// TIA Portal V18 export
FUNCTION "Ratio Check Program sequences" : Void   // FC6, LAD
{ S7_Optimized_Access := 'TRUE' }
VERSION : 0.1
// stored: AutoNumber true, IsIECCheckEnabled false, SetENOAutomatically false, UDAEnableTagReadback false
   VAR_TEMP
      temp1 : Bool;
   END_VAR
   VAR_TEMP   // added for the SCL form of the ladder/FBD networks
      _w1 : Bool;
      _w2 : Bool;
      _w3 : Bool;
      _w4 : Bool;
   END_VAR
BEGIN

REGION Network 1
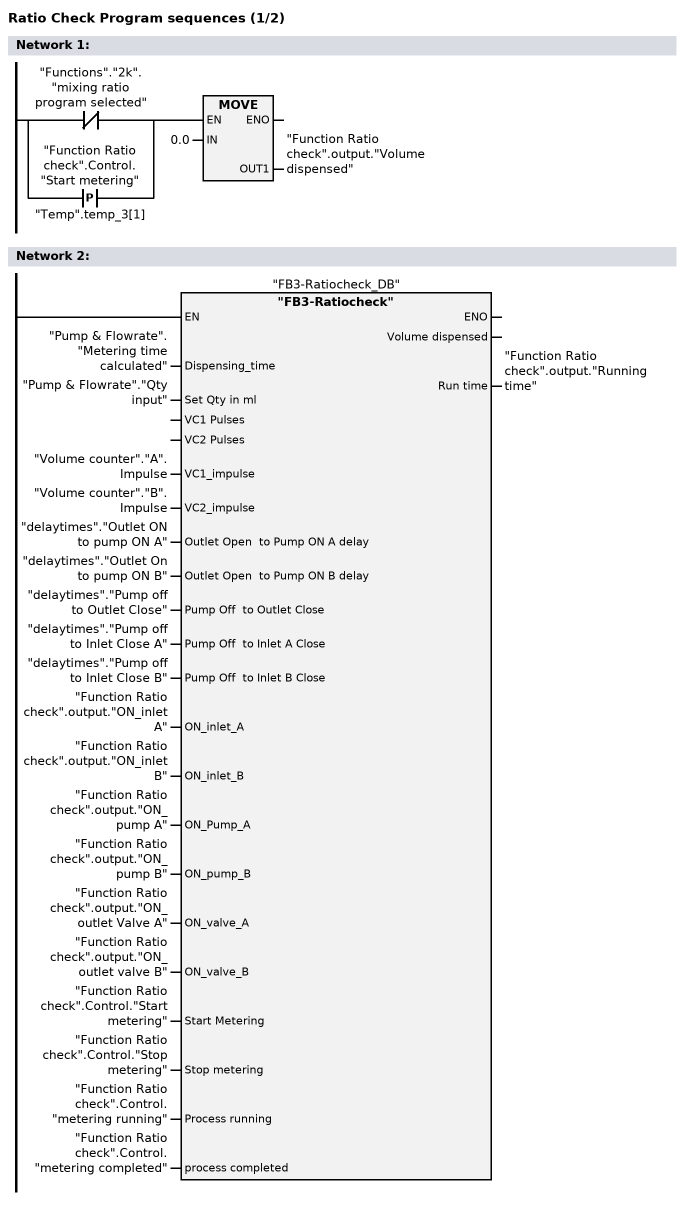
   RUNG wire#powerrail
      I_Contact( "Functions"."2k"."mixing ratio program selected" )
      wire#w1
      Move(in := 0.0, out1 => "Function Ratio check".output."Volume dispensed")
   END_RUNG
   RUNG wire#powerrail
      P_Contact(operand := "Function Ratio check".Control."Start metering", bit := "Temp".temp_3[1])
   END_RUNG wire#w1
   // the same network as SCL:
   #_w1 := "Function Ratio check".Control."Start metering" AND NOT "Temp".temp_3[1];   // rising edge of "Function Ratio check".Control."Start metering"
   "Temp".temp_3[1] := "Function Ratio check".Control."Start metering";
   IF NOT "Functions"."2k"."mixing ratio program selected" OR #_w1 THEN
       "Function Ratio check".output."Volume dispensed" := 0.0;
   END_IF;
END_REGION

REGION Network 2
   RUNG wire#powerrail
      "FB3-Ratiocheck_DB"(Dispensing_time := "Pump & Flowrate"."Metering time calculated", "Set Qty in ml" := "Pump & Flowrate"."Qty input", "VC1 Pulses" :=, "VC2 Pulses" :=, VC1_impulse := "Volume counter"."A".Impulse, VC2_impulse := "Volume counter"."B".Impulse, "Outlet Open  to Pump ON A delay" := "delaytimes"."Outlet ON to pump ON A", "Outlet Open  to Pump ON B delay" := "delaytimes"."Outlet On to pump ON B", "Pump Off  to Outlet Close" := "delaytimes"."Pump off to Outlet Close", "Pump Off  to Inlet A Close" := "delaytimes"."Pump off to Inlet Close A", "Pump Off  to Inlet B Close" := "delaytimes"."Pump off to Inlet Close B", ON_inlet_A := "Function Ratio check".output."ON_inlet A", ON_inlet_B := "Function Ratio check".output."ON_inlet B", ON_Pump_A := "Function Ratio check".output."ON_pump A", ON_pump_B := "Function Ratio check".output."ON_pump B", ON_valve_A := "Function Ratio check".output."ON_outlet Valve A", ON_valve_B := "Function Ratio check".output."ON_outlet valve B", "Start Metering" := "Function Ratio check".Control."Start metering", "Stop metering" := "Function Ratio check".Control."Stop metering", "Process running" := "Function Ratio check".Control."metering running", "process completed" := "Function Ratio check".Control."metering completed", "Volume dispensed" =>, "Run time" => "Function Ratio check".output."Running time")
   END_RUNG
   // the same network as SCL:
   "FB3-Ratiocheck_DB"(Dispensing_time := "Pump & Flowrate"."Metering time calculated",   // "FB3-Ratiocheck"
                       "Set Qty in ml" := "Pump & Flowrate"."Qty input",
                       VC1_impulse := "Volume counter"."A".Impulse,
                       VC2_impulse := "Volume counter"."B".Impulse,
                       "Outlet Open  to Pump ON A delay" := "delaytimes"."Outlet ON to pump ON A",
                       "Outlet Open  to Pump ON B delay" := "delaytimes"."Outlet On to pump ON B",
                       "Pump Off  to Outlet Close" := "delaytimes"."Pump off to Outlet Close",
                       "Pump Off  to Inlet A Close" := "delaytimes"."Pump off to Inlet Close A",
                       "Pump Off  to Inlet B Close" := "delaytimes"."Pump off to Inlet Close B",
                       ON_inlet_A := "Function Ratio check".output."ON_inlet A",
                       ON_inlet_B := "Function Ratio check".output."ON_inlet B",
                       ON_Pump_A := "Function Ratio check".output."ON_pump A",
                       ON_pump_B := "Function Ratio check".output."ON_pump B",
                       ON_valve_A := "Function Ratio check".output."ON_outlet Valve A",
                       ON_valve_B := "Function Ratio check".output."ON_outlet valve B",
                       "Start Metering" := "Function Ratio check".Control."Start metering",
                       "Stop metering" := "Function Ratio check".Control."Stop metering",
                       "Process running" := "Function Ratio check".Control."metering running",
                       "process completed" := "Function Ratio check".Control."metering completed",
                       "Run time" => "Function Ratio check".output."Running time");
END_REGION

REGION Network 3: Volume dispensed
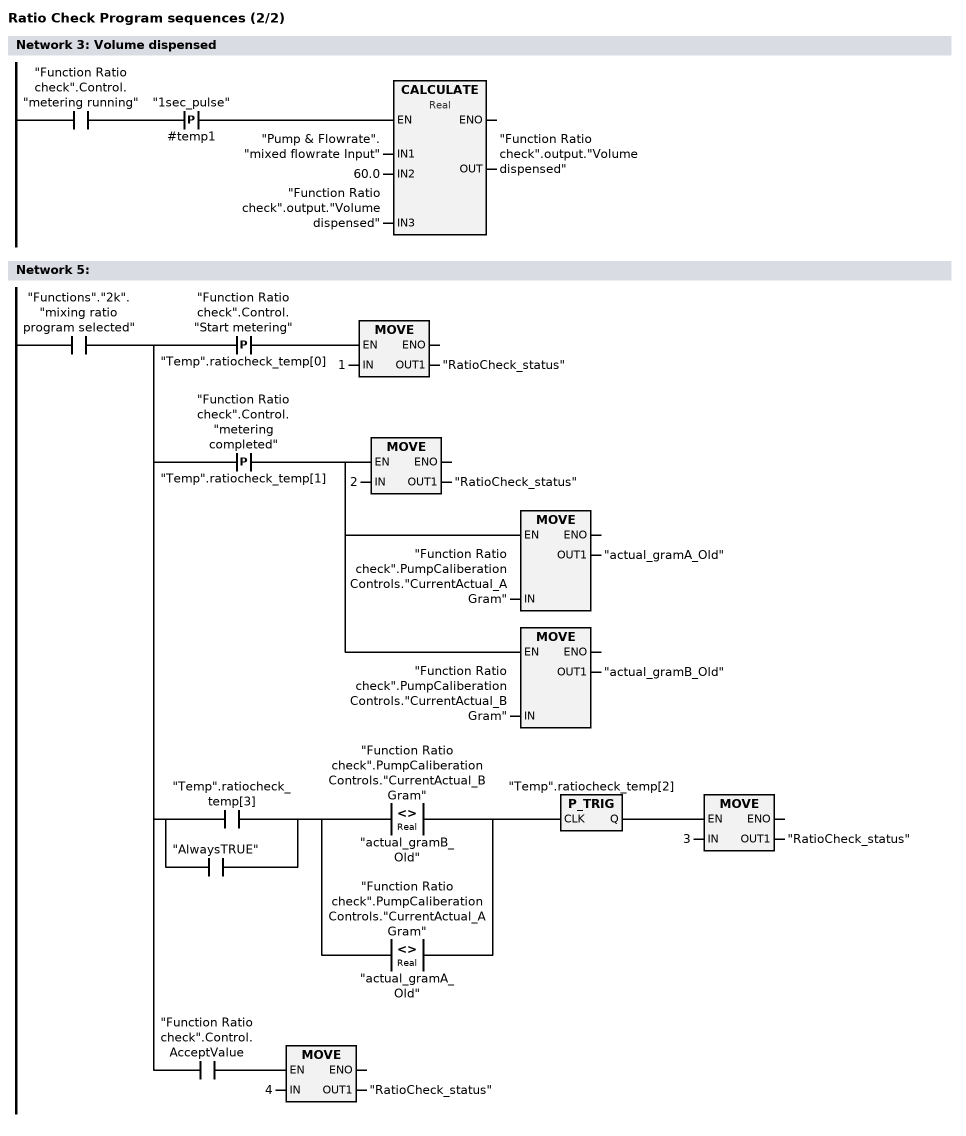
   RUNG wire#powerrail
      Contact( "Function Ratio check".Control."metering running" )
      P_Contact(operand := "1sec_pulse", bit := #temp1)
      { S7_Templates := "SrcType := Real"; S7_Expression := "(IN1/IN2)+IN3" } Calculate(in1 := "Pump & Flowrate"."mixed flowrate Input", in2 := 60.0, in3 := "Function Ratio check".output."Volume dispensed", out => "Function Ratio check".output."Volume dispensed")
   END_RUNG
   // the same network as SCL:
   #_w1 := "Function Ratio check".Control."metering running" AND "1sec_pulse" AND NOT #temp1;   // rising edge of "1sec_pulse"
   #temp1 := "1sec_pulse";
   IF #_w1 THEN
       "Function Ratio check".output."Volume dispensed" := ("Pump & Flowrate"."mixed flowrate Input"/60.0)+"Function Ratio check".output."Volume dispensed";
   END_IF;
END_REGION

REGION Network 5
   RUNG wire#powerrail
      Contact( "Functions"."2k"."mixing ratio program selected" )
      wire#w1
      P_Contact(operand := "Function Ratio check".Control."Start metering", bit := "Temp".ratiocheck_temp[0])
      Move(in := 1, out1 => "RatioCheck_status")
   END_RUNG
   RUNG wire#w1
      P_Contact(operand := "Function Ratio check".Control."metering completed", bit := "Temp".ratiocheck_temp[1])
      wire#w2
      Move(in := 2, out1 => "RatioCheck_status")
   END_RUNG
   RUNG wire#w2
      Move(in := "Function Ratio check".PumpCaliberationControls."CurrentActual_A Gram", out1 => "actual_gramA_Old")
   END_RUNG
   RUNG wire#w2
      Move(in := "Function Ratio check".PumpCaliberationControls."CurrentActual_B Gram", out1 => "actual_gramB_Old")
   END_RUNG
   RUNG wire#w1
      Contact( "Temp".ratiocheck_temp[3] )
      wire#w3
      { S7_Templates := "SrcType := Real" } NE_Contact(in1 := "Function Ratio check".PumpCaliberationControls."CurrentActual_B Gram", in2 := "actual_gramB_Old")
      wire#w4
      P_Trig( "Temp".ratiocheck_temp[2] )
      Move(in := 3, out1 => "RatioCheck_status")
   END_RUNG
   RUNG wire#w1
      Contact( "AlwaysTRUE" )
   END_RUNG wire#w3
   RUNG wire#w3
      { S7_Templates := "SrcType := Real" } NE_Contact(in1 := "Function Ratio check".PumpCaliberationControls."CurrentActual_A Gram", in2 := "actual_gramA_Old")
   END_RUNG wire#w4
   RUNG wire#w1
      Contact( "Function Ratio check".Control.AcceptValue )
      Move(in := 4, out1 => "RatioCheck_status")
   END_RUNG
   // the same network as SCL:
   #_w1 := "Functions"."2k"."mixing ratio program selected" AND "Function Ratio check".Control."Start metering" AND NOT "Temp".ratiocheck_temp[0];   // rising edge of "Function Ratio check".Control."Start metering"
   "Temp".ratiocheck_temp[0] := "Function Ratio check".Control."Start metering";
   IF #_w1 THEN "RatioCheck_status" := 1; END_IF;
   #_w2 := "Functions"."2k"."mixing ratio program selected" AND "Function Ratio check".Control."metering completed" AND NOT "Temp".ratiocheck_temp[1];   // rising edge of "Function Ratio check".Control."metering completed"
   "Temp".ratiocheck_temp[1] := "Function Ratio check".Control."metering completed";
   IF #_w2 THEN
       "RatioCheck_status" := 2;
       "actual_gramA_Old" := "Function Ratio check".PumpCaliberationControls."CurrentActual_A Gram";
       "actual_gramB_Old" := "Function Ratio check".PumpCaliberationControls."CurrentActual_B Gram";
   END_IF;
   #_w3 := "Functions"."2k"."mixing ratio program selected" AND ("Temp".ratiocheck_temp[3] OR "AlwaysTRUE") AND (("Function Ratio check".PumpCaliberationControls."CurrentActual_B Gram" <> "actual_gramB_Old") OR ("Function Ratio check".PumpCaliberationControls."CurrentActual_A Gram" <> "actual_gramA_Old"));
   #_w4 := #_w3 AND NOT "Temp".ratiocheck_temp[2];   // rising edge
   "Temp".ratiocheck_temp[2] := #_w3;
   IF #_w4 THEN "RatioCheck_status" := 3; END_IF;
   IF "Functions"."2k"."mixing ratio program selected" AND "Function Ratio check".Control.AcceptValue THEN
       "RatioCheck_status" := 4;
   END_IF;
END_REGION
END_FUNCTION
